// TIA Portal V19 export
FUNCTION "FC_SIMULATION" : Void   // FC200, STL
TITLE = SIMULATION
{ S7_Optimized_Access := 'FALSE' }
AUTHOR : RE
// stored: AutoNumber false
   VAR_TEMP
      count : Int;
      AnzahlWT : Int;
      Faktor : Real;
      TR3 : Real;
      ErrInf : Byte;
      ON : Bool;
      OFF : Bool;
      dummy : Bool;
      Takt : Bool;
      BE_Auto : Bool;
      low : Bool;
      "return" : Bool;
      S01 : Bool;
      S02 : Bool;
      S03 : Bool;
      S04 : Bool;
      S05 : Bool;
      S06 : Bool;
      S07 : Bool;
      S00 : Bool;
      HZ1 : Bool;   // Heizung 1 an
      HZ2 : Bool;   // Heizung 2 an
      KHL : Bool;   // Kühlung an
      TypExo : Bool;   // Bad mit Kühlregler
      v0 : Bool;
   END_VAR
BEGIN

NETWORK
TITLE = Simulation Anlage

      AN    "DB_ANLAGE".BA.Simulation;
      BEC;

//-------------------------
//Beladestände simulieren
//-------------------------
      L     "DB_POS".POS[25].WT_DB;
      L     0;
      <>I;
      S     "DB_BE_Stand".Stand[1].IN_Belegt;

      A     "DB_POS".POS[25].FW_Hebt;
      AN    "DI_FW_1".ZST.low_SU_li;
      R     "DB_BE_Stand".Stand[1].IN_Belegt;

      SET;
      =     "DB_BE_Stand".Stand[1].IN_innen;
      =     "DB_BE_Stand".Stand[1].IN_aussen;
      =     "DB_BE_Stand".Stand[1].verriegelt;
      =     "DB_BE_Stand".Stand[1].IN_Freigabe;

      L     "DB_POS".POS[26].WT_DB;
      L     0;
      <>I;
      S     "DB_BE_Stand".Stand[2].IN_Belegt;

      A     "DB_POS".POS[26].FW_Hebt;
      AN    "DI_FW_1".ZST.low_SU_re;
      R     "DB_BE_Stand".Stand[2].IN_Belegt;

      SET;
      =     "DB_BE_Stand".Stand[2].IN_innen;
      =     "DB_BE_Stand".Stand[2].IN_aussen;
      =     "DB_BE_Stand".Stand[2].verriegelt;
      =     "DB_BE_Stand".Stand[2].IN_Freigabe;

      L     "DB_POS".POS[27].WT_DB;
      L     0;
      <>I;
      S     "DB_BE_Stand".Stand[3].IN_Belegt;

      A     "DB_POS".POS[27].FW_Hebt;
      AN    "DI_FW_1".ZST.low_SU_li;
      R     "DB_BE_Stand".Stand[3].IN_Belegt;

      SET;
      =     "DB_BE_Stand".Stand[3].IN_innen;
      =     "DB_BE_Stand".Stand[3].IN_aussen;
      =     "DB_BE_Stand".Stand[3].verriegelt;
      =     "DB_BE_Stand".Stand[3].IN_Freigabe;

      L     "DB_POS".POS[28].WT_DB;
      L     0;
      <>I;
      S     "DB_BE_Stand".Stand[2].IN_Belegt;

      A     "DB_POS".POS[28].FW_Hebt;
      AN    "DI_FW_1".ZST.low_SU_re;
      R     "DB_BE_Stand".Stand[4].IN_Belegt;

      SET;
      =     "DB_BE_Stand".Stand[4].IN_innen;
      =     "DB_BE_Stand".Stand[4].IN_aussen;
      =     "DB_BE_Stand".Stand[4].verriegelt;
      =     "DB_BE_Stand".Stand[4].IN_Freigabe;

      L     "DB_POS".POS[29].WT_DB;
      L     0;
      <>I;
      S     "DB_BE_Stand".Stand[5].IN_Belegt;

      A     "DB_POS".POS[29].FW_Hebt;
      AN    "DI_FW_1".ZST.low_SU_li;
      R     "DB_BE_Stand".Stand[5].IN_Belegt;

      SET;
      =     "DB_BE_Stand".Stand[5].IN_innen;
      =     "DB_BE_Stand".Stand[5].IN_aussen;
      =     "DB_BE_Stand".Stand[5].verriegelt;
      =     "DB_BE_Stand".Stand[5].IN_Freigabe;

      L     "DB_POS".POS[30].WT_DB;
      L     0;
      <>I;
      S     "DB_BE_Stand".Stand[6].IN_Belegt;

      A     "DB_POS".POS[30].FW_Hebt;
      AN    "DI_FW_1".ZST.low_SU_re;
      R     "DB_BE_Stand".Stand[6].IN_Belegt;

      SET;
      =     "DB_BE_Stand".Stand[6].IN_innen;
      =     "DB_BE_Stand".Stand[6].IN_aussen;
      =     "DB_BE_Stand".Stand[6].verriegelt;
      =     "DB_BE_Stand".Stand[6].IN_Freigabe;



NETWORK
TITLE = Transportsystem
//****************************************
//           Transportsystem
//****************************************
      L     S5T#2S;
      A     "DB_ANLAGE".IN.S_Not_Aus;
      SF    "T_Verz_NotAus";

      SET;
      =     "DI_FW_1".IN.Laser_on;

//------------------------------------
//             Fahrwagen 1
//------------------------------------
      SET;
      =     "DI_FW_1".IN.Laser_on;

//Stellung Unten
      L     "DI_FW_1".ZST.HubInc_li;
      L     "DI_FW_1".PAR.Hub.Ebene0;
      -D;
      DTR;
      ABS;
      RND;
      L     "DI_FW_1".PAR.Hub.Bereich_Pos;
      <=D;
      =     "DI_FW_1".IN.Unten_li;

//Stellung oben
      L     "DI_FW_1".ZST.HubInc_li;
      L     "DI_FW_1".PAR.Hub.Ebene3;
      -D;
      DTR;
      ABS;
      RND;
      L     "DI_FW_1".PAR.Hub.Bereich_Pos;
      <=D;
      =     "DI_FW_1".IN.Oben_li;

//Stellung Unten
      L     "DI_FW_1".HELP.HubInc_re;
      L     "DI_FW_1".PAR.Hub.Ebene0;
      -D;
      DTR;
      ABS;
      RND;
      L     "DI_FW_1".PAR.Hub.Bereich_Pos;
      <=D;
      =     "DI_FW_1".IN.Unten_re;

//Stellung oben
      L     "DI_FW_1".HELP.HubInc_re;
      L     "DI_FW_1".PAR.Hub.Ebene3;
      -D;
      DTR;
      ABS;
      RND;
      L     "DI_FW_1".PAR.Hub.Bereich_Pos;
      <=D;
      =     "DI_FW_1".IN.Oben_re;

END_FUNCTION
